FUNCTION_BLOCK Blinker
VAR_INPUT
	Taktzeit: TIME;
END_VAR
VAR_OUTPUT
	Ausgang: BOOL;
END_VAR
VAR
	Timer1: TON;
END_VAR

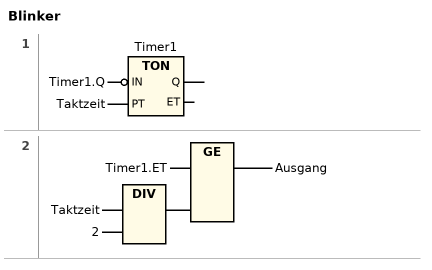
// NETWORK 1
Timer1(IN := NOT Timer1.Q, PT := Taktzeit); // TON

// NETWORK 2
Ausgang := Timer1.ET >= Taktzeit / 2;

END_FUNCTION_BLOCK

(* stored: Version 1.1.0.1, ProductVersion 3.1.0.12
   POU Blinker: Id {fdc6f2a4-9c0b-4322-9634-38882faa3f8c} *)
